Fanuc KAREL source: kt00982.KL

-- PROVISIONAL review KL for V770-1; original PC SHA256 2754e140d69678581b87101098c6717c80814fe26e919809d4416aadc4d38f4a
-- Incomplete behavior may be omitted. Consult companion uncertainty JSON. Do not deploy.
PROGRAM KT00982
%NOLOCKGROUP
VAR
  R1 : REAL
  R2 : REAL
-- UNRESOLVED_DECL CFG type=00001c
-- UNRESOLVED_DECL OUT type=000101
BEGIN
  -- UNRESOLVED_PC offsets 5-16; opcodes 2E,23
  -- UNRESOLVED_PC offsets 21-32; opcodes 2E,23
  -- UNRESOLVED_PC offsets 37-48; opcodes 2E,23
  -- UNRESOLVED_PC offsets 53-64; opcodes 2E,23
  -- UNRESOLVED_PC offsets 69-79; opcodes 9D,22,A5
  -- UNRESOLVED_PC offsets 84-141; opcodes 27,22,22,22,22,22,22,22,76,7E,4A
  -- UNRESOLVED_PC offsets 146-150; opcodes 7F
END KT00982
